// Mitsubishi GX Works2 project: PLC_Group_05 (1)   PLC: FX3G

// global labels: Global1
VAR_GLOBAL
  StartDay AT X007 : BOOL;
  StartCycle AT X001 : BOOL;
  StartCooling AT X002 : BOOL;
  TempSensor AT X003 : BOOL;
  EmergencyStop AT X005 : BOOL;
  WorkDayLamp AT Y007 : BOOL;
  FlavorLamp AT Y000 : BOOL;
  CoolingMotor AT Y002 : BOOL;
  MixLampA AT Y005 : BOOL;
  MixLampB AT Y006 : BOOL;
  StockError AT M0 : BOOL;
  SampleError AT M1 : BOOL;
  RegularPk AT M11 : BOOL;
  PremiumPk AT M12 : BOOL;
  CoolingDone AT M22 : BOOL;
  MixingDone AT M23 : BOOL;
  Flicker AT M30 : BOOL;
  DayEnd AT M40 : BOOL;
  InCycle AT M50 : BOOL;
  MixingActive AT M60 : BOOL;
END_VAR
VAR_GLOBAL CONSTANT
  RaspReg : REAL := 280;
  LemonReg : REAL := 455;
  SolidReg : REAL := 105;
  GummyReg : REAL := 28;
  RaspPm : REAL := 385;
  LemonPm : REAL := 665;
  SolidPm : REAL := 210;
  GummyPm : REAL := 70;
  RCreamReg : REAL := 350;
  LCreamReg : REAL := 490;
  RCreamPm : REAL := 560;
  LCreamPm : REAL := 700;
END_VAR
VAR_GLOBAL
  InitialRasp AT D1110 : REAL;
  Raspberry AT D1100 : REAL;
  InitialLemon AT D1112 : REAL;
  Lemon AT D1102 : REAL;
  InitialSolid AT D1114 : REAL;
  Solidifier AT D1104 : REAL;
  InitialGummy AT D1116 : REAL;
  GummyBears AT D1106 : REAL;
  AnalogIn AT D8280 : INT;
  Sample AT D1506 : REAL;
  FlavorsDone AT M21 : BOOL;
  RaspTank AT D1200 : REAL;
  LemonTank AT D1202 : REAL;
  Time2 AT TC2 : BOOL;
  Time1 AT TC1 : BOOL;
END_VAR
VAR_GLOBAL CONSTANT
  CoolingTime : INT := K80;
  FlavorsTime : INT := K50;
END_VAR
VAR_GLOBAL
  TS_2 AT TS2 : BOOL;
  TS_1 AT TS1 : BOOL;
  MixTank AT D1204 : REAL;
  Time3 AT TC3 : BOOL;
  Time4 AT TC4 : BOOL;
  TS_4 AT TS4 : BOOL;
  Time5 AT TC5 : BOOL;
  TS_5 AT TS5 : BOOL;
  PkCounter AT CC1 : BOOL;
  AnalogOut AT D8282 : INT;
  TS_3 AT TS3 : BOOL;
END_VAR
VAR_GLOBAL CONSTANT
  ResetZero : REAL;
END_VAR
VAR_GLOBAL
  SaveAnalog AT D8200 : INT;
  SampledFlag AT M2 : BOOL;
  RegularLack AT M111 : BOOL;
  PremiumLack AT M122 : BOOL;
  CS_1 AT CS1 : BOOL;
  InventoryToday AT D7996 : REAL;
  MixTime AT D8004 : INT;
  SubComplete AT M51 : BOOL;
END_VAR
VAR_GLOBAL CONSTANT
  MixTimeReg : INT := 30;
  MixTimePre : INT := 50;
END_VAR
VAR_GLOBAL
  Time3_1 AT TC6 : BOOL;
  TS_3_1 AT TS6 : BOOL;
  CycleDone AT M24 : BOOL;
END_VAR

// task Task_01 (event TRUE, interval 0, priority 31): POU_01

PROGRAM POU_01
(* structured ladder/FBD written out as ST: instructions are called as NAME(EN, inputs, outputs); _pN, _eN, _tN stand for wires *)
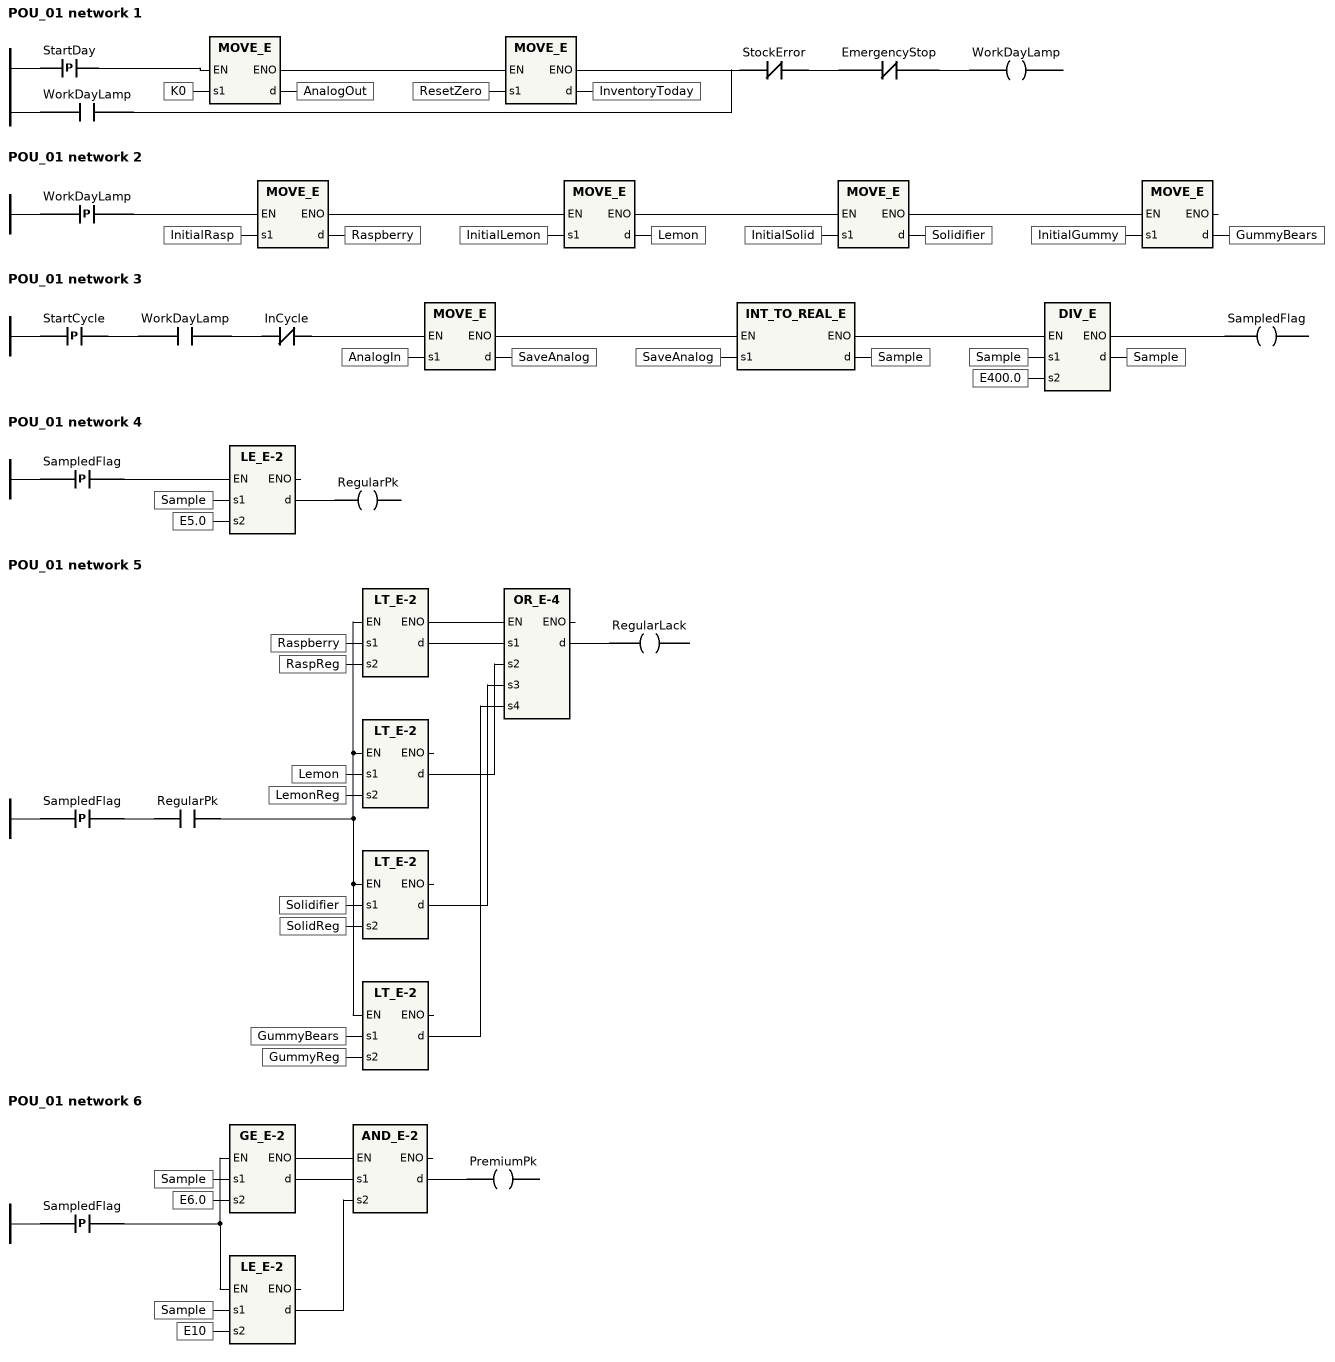
(* network 1 *)
_e1 := MOVE_E(LDP(TRUE, StartDay), K0, AnalogOut);
_e2 := MOVE_E(_e1, ResetZero, InventoryToday);
WorkDayLamp := ((_e2 OR WorkDayLamp) AND NOT StockError) AND NOT EmergencyStop;
(* network 2 *)
_e1 := MOVE_E(LDP(TRUE, WorkDayLamp), InitialRasp, Raspberry);
_e2 := MOVE_E(_e1, InitialLemon, Lemon);
_e3 := MOVE_E(_e2, InitialSolid, Solidifier);
MOVE_E(_e3, InitialGummy, GummyBears);
(* network 3 *)
_e1 := MOVE_E(LDP(TRUE, StartCycle) AND WorkDayLamp AND NOT InCycle, AnalogIn, SaveAnalog);
_e2 := INT_TO_REAL_E(_e1, SaveAnalog, Sample);
_e3 := DIV_E(_e2, Sample, E400.0, Sample);
SampledFlag := _e3;
(* network 4 *)
LE_E(LDP(TRUE, SampledFlag), Sample, E5.0, _t1);
RegularPk := _t1;
(* network 5 *)
_p1 := LDP(TRUE, SampledFlag) AND RegularPk;
_e3 := LT_E(_p1, Raspberry, RaspReg, _t2);
LT_E(_p1, Lemon, LemonReg, _t4);
LT_E(_p1, Solidifier, SolidReg, _t5);
LT_E(_p1, GummyBears, GummyReg, _t6);
OR_E(_e3, _t2, _t4, _t5, _t6, _t7);
RegularLack := _t7;
(* network 6 *)
_p1 := LDP(TRUE, SampledFlag);
_e3 := GE_E(_p1, Sample, E6.0, _t2);
LE_E(_p1, Sample, E10, _t4);
AND_E(_e3, _t2, _t4, _t5);
PremiumPk := _t5;
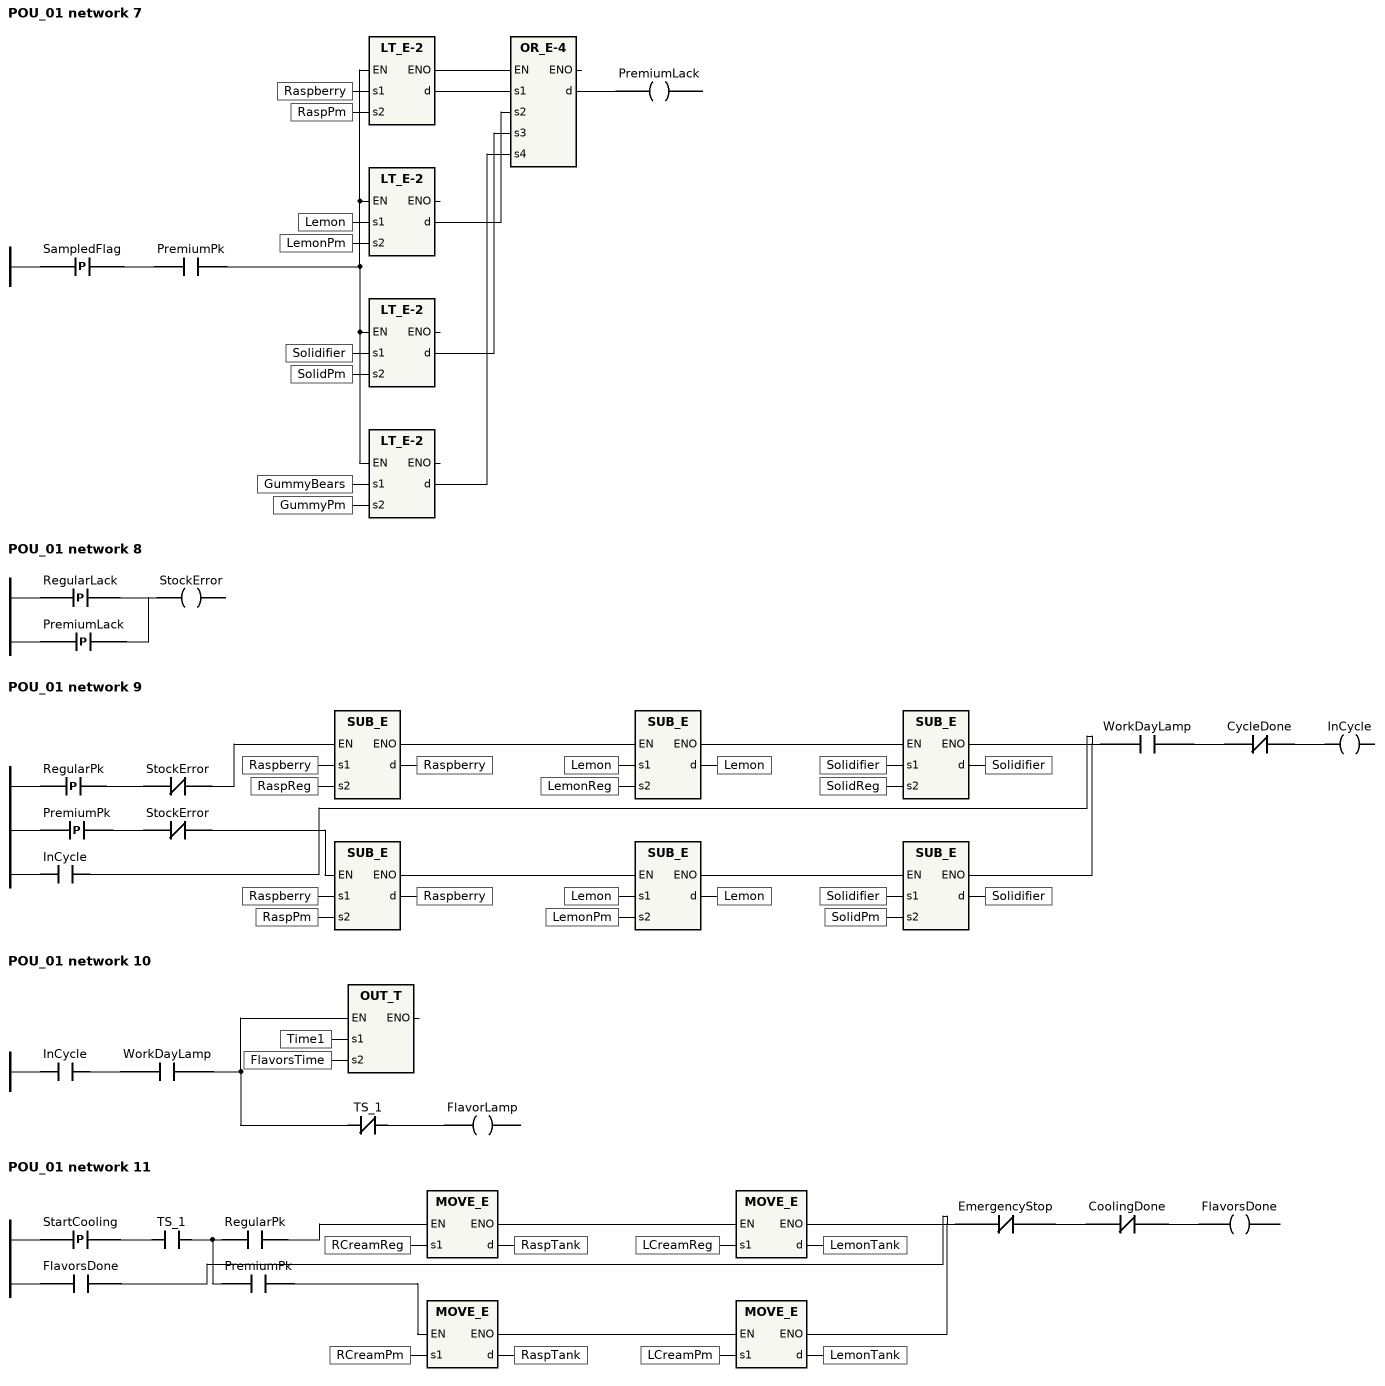
(* network 7 *)
_p1 := LDP(TRUE, SampledFlag) AND PremiumPk;
_e3 := LT_E(_p1, Raspberry, RaspPm, _t2);
LT_E(_p1, Lemon, LemonPm, _t4);
LT_E(_p1, Solidifier, SolidPm, _t5);
LT_E(_p1, GummyBears, GummyPm, _t6);
OR_E(_e3, _t2, _t4, _t5, _t6, _t7);
PremiumLack := _t7;
(* network 8 *)
StockError := LDP(TRUE, RegularLack) OR LDP(TRUE, PremiumLack);
(* network 9 *)
_e1 := SUB_E(LDP(TRUE, RegularPk) AND NOT StockError, Raspberry, RaspReg, Raspberry);
_e2 := SUB_E(_e1, Lemon, LemonReg, Lemon);
_e3 := SUB_E(_e2, Solidifier, SolidReg, Solidifier);
_e4 := SUB_E(LDP(TRUE, PremiumPk) AND NOT StockError, Raspberry, RaspPm, Raspberry);
_e5 := SUB_E(_e4, Lemon, LemonPm, Lemon);
_e6 := SUB_E(_e5, Solidifier, SolidPm, Solidifier);
InCycle := ((_e3 OR _e6 OR InCycle) AND WorkDayLamp) AND NOT CycleDone;
(* network 10 *)
_p1 := InCycle AND WorkDayLamp;
OUT_T(_p1, Time1, FlavorsTime);
FlavorLamp := _p1 AND NOT TS_1;
(* network 11 *)
_p1 := LDP(TRUE, StartCooling) AND TS_1;
_e2 := MOVE_E(_p1 AND RegularPk, RCreamReg, RaspTank);
_e3 := MOVE_E(_e2, LCreamReg, LemonTank);
_e4 := MOVE_E(_p1 AND PremiumPk, RCreamPm, RaspTank);
_e5 := MOVE_E(_e4, LCreamPm, LemonTank);
FlavorsDone := ((_e3 OR _e5 OR FlavorsDone) AND NOT EmergencyStop) AND NOT CoolingDone;
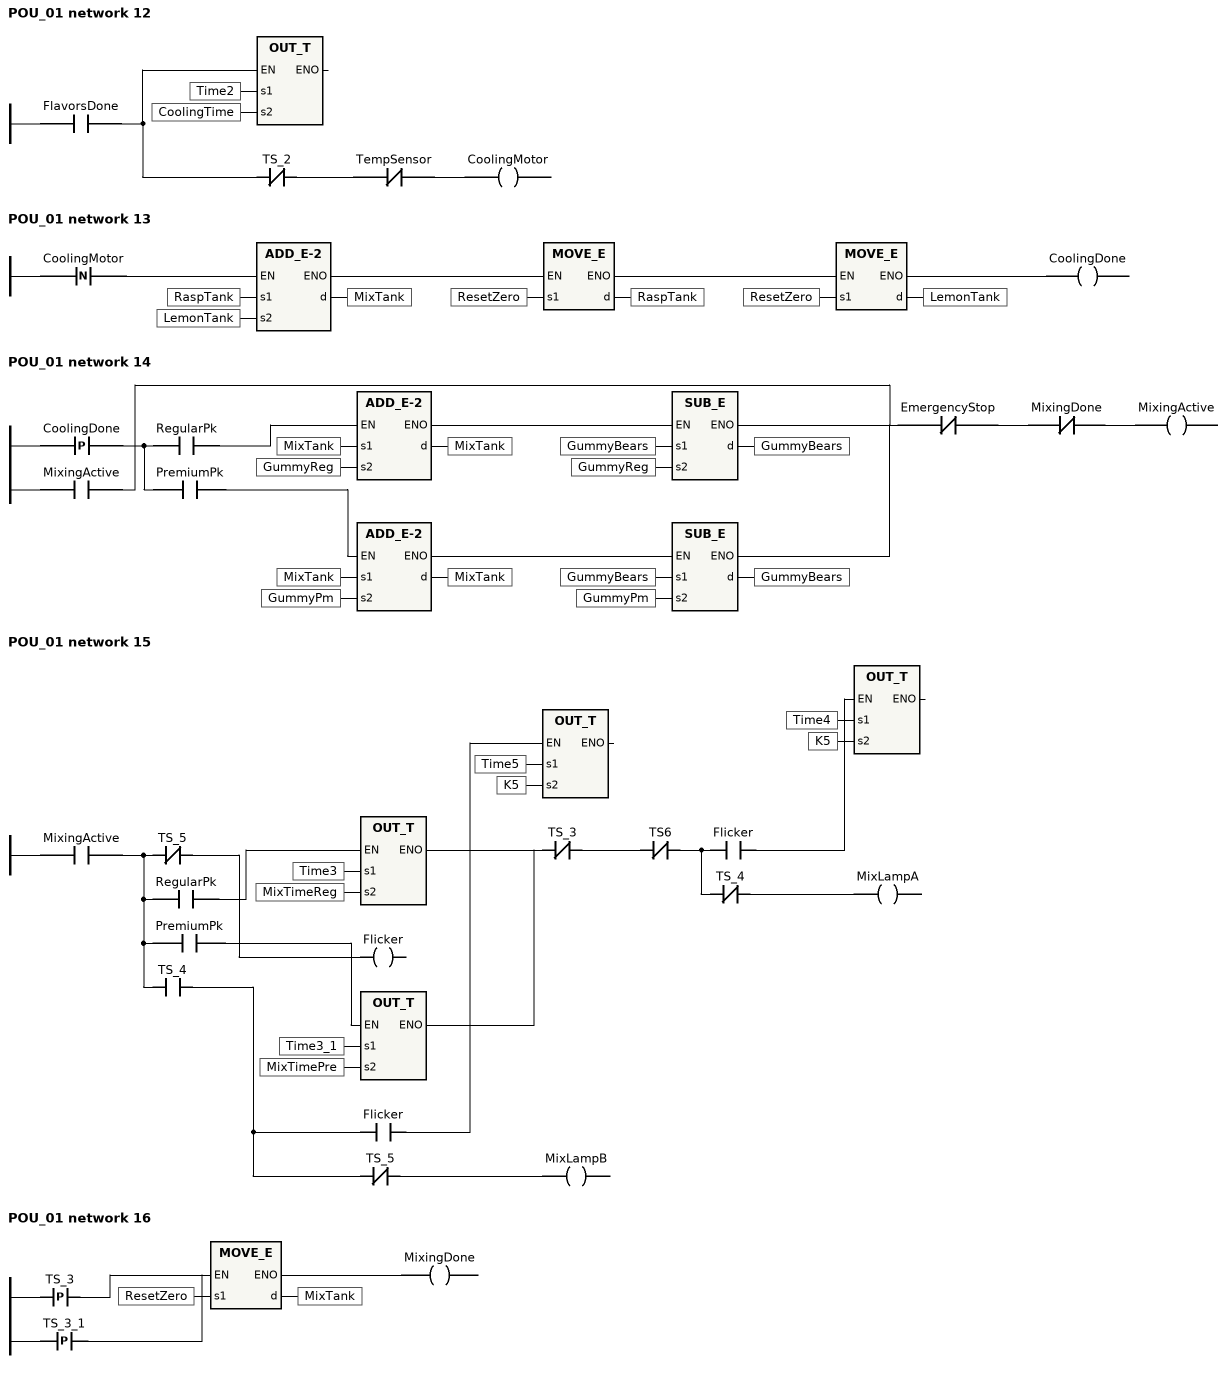
(* network 12 *)
OUT_T(FlavorsDone, Time2, CoolingTime);
CoolingMotor := FlavorsDone AND NOT TS_2 AND NOT TempSensor;
(* network 13 *)
_e1 := ADD_E(LDF(TRUE, CoolingMotor), RaspTank, LemonTank, MixTank);
_e2 := MOVE_E(_e1, ResetZero, RaspTank);
_e3 := MOVE_E(_e2, ResetZero, LemonTank);
CoolingDone := _e3;
(* network 14 *)
_p1 := LDP(TRUE, CoolingDone);
_e2 := ADD_E(_p1 AND RegularPk, MixTank, GummyReg, MixTank);
_e3 := SUB_E(_e2, GummyBears, GummyReg, GummyBears);
_e4 := ADD_E(_p1 AND PremiumPk, MixTank, GummyPm, MixTank);
_e5 := SUB_E(_e4, GummyBears, GummyPm, GummyBears);
MixingActive := ((_e3 OR _e5 OR MixingActive) AND NOT EmergencyStop) AND NOT MixingDone;
(* network 15 *)
Flicker := MixingActive AND NOT TS_5;
_e1 := OUT_T(MixingActive AND RegularPk, Time3, MixTimeReg);
_e2 := OUT_T(MixingActive AND PremiumPk, Time3_1, MixTimePre);
_p3 := ((_e1 OR _e2) AND NOT TS_3) AND NOT TS6;
OUT_T(_p3 AND Flicker, Time4, K5);
MixLampA := _p3 AND NOT TS_4;
_p4 := MixingActive AND TS_4;
OUT_T(_p4 AND Flicker, Time5, K5);
MixLampB := _p4 AND NOT TS_5;
(* network 16 *)
_e1 := MOVE_E(LDP(TRUE, TS_3) OR LDP(TRUE, TS_3_1), ResetZero, MixTank);
MixingDone := _e1;
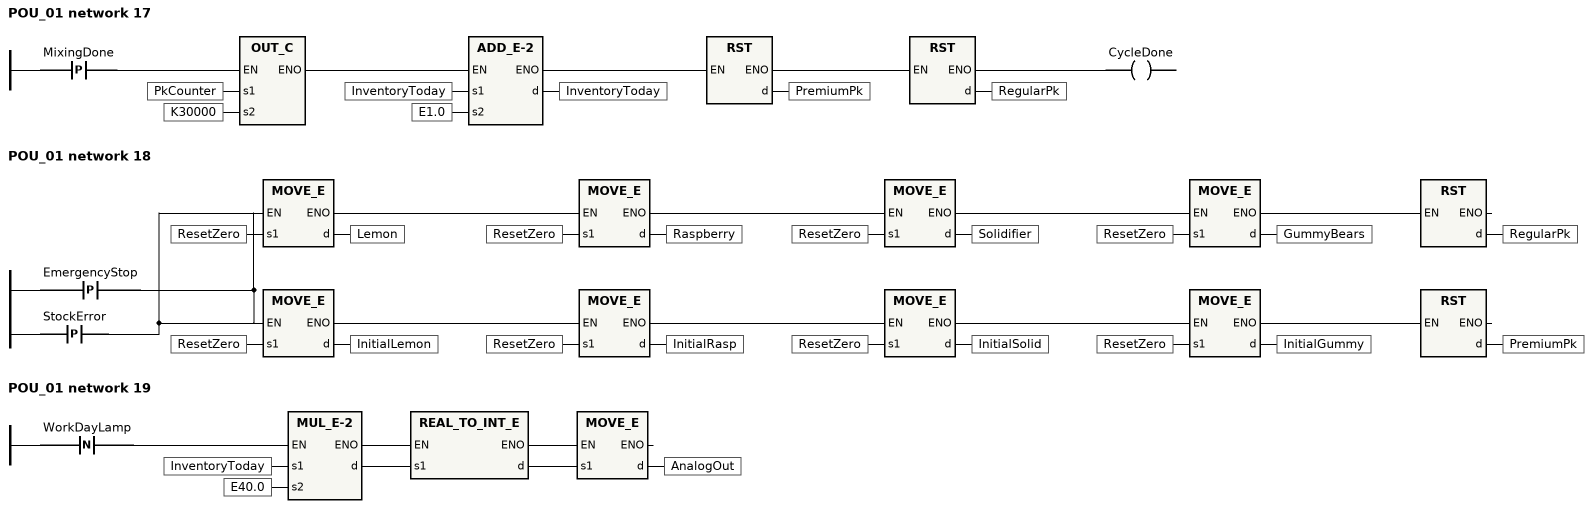
(* network 17 *)
_e1 := OUT_C(LDP(TRUE, MixingDone), PkCounter, K30000);
_e2 := ADD_E(_e1, InventoryToday, E1.0, InventoryToday);
_e3 := RST(_e2, PremiumPk);
_e4 := RST(_e3, RegularPk);
CycleDone := _e4;
(* network 18 *)
_p1 := LDP(TRUE, EmergencyStop) OR LDP(TRUE, StockError);
_e2 := MOVE_E(_p1, ResetZero, Lemon);
_e3 := MOVE_E(_e2, ResetZero, Raspberry);
_e4 := MOVE_E(_e3, ResetZero, Solidifier);
_e5 := MOVE_E(_e4, ResetZero, GummyBears);
RST(_e5, RegularPk);
_e6 := MOVE_E(_p1, ResetZero, InitialLemon);
_e7 := MOVE_E(_e6, ResetZero, InitialRasp);
_e8 := MOVE_E(_e7, ResetZero, InitialSolid);
_e9 := MOVE_E(_e8, ResetZero, InitialGummy);
RST(_e9, PremiumPk);
(* network 19 *)
_e2 := MUL_E(LDF(TRUE, WorkDayLamp), InventoryToday, E40.0, _t1);
_e4 := REAL_TO_INT_E(_e2, _t1, _t3);
MOVE_E(_e4, _t3, AnalogOut);
END_PROGRAM
